{attribute 'qualified_only'}
{attribute 'strict'}
{attribute 'to_string'}
TYPE E_WaferHandlingType :
(
	Unknown := 0,
	Passive,
	Active
);
END_TYPE

(* stored: Version 1.1.0.1, ProductVersion 3.1.4026.18
   DUT E_WaferHandlingType: Id {424faf8f-29b5-4329-8407-b61d38aba62b} *)
